// SIMATIC S7-200 project (STEP 7-Micro/WIN), CPU 226 CN REL 02.01

ORGANIZATION_BLOCK 主程序:OB1
TITLE=程序是控制时效炉，用于金属材料热处理
// 
// 风机启动前应确认风压正常。通过风机启动触发鼓风机启动，但鼓风机启动前必须确认东门下限和西门下限已关闭且无故障光报警，以确保通风正常，避免因风压不足影响热处理效果。
// 风机启动后，利用星转角时间切换至风机运行，提供稳定的炉内空气循环。
// 风机运行时，风压开关检测风压状态，若风压异常则触发无风压检测。
// 随后，东门上升和东门下降控制门的位置，但东门上升或东门下降时，必须确认东车运行中为假且未到达东门上限或东门下限，防止门与车碰撞或超出行程。
// 接着，东车前进将材料送入炉内，而东车前进或东车后退时，必须确认东门放松限位为真且无故障光报警，确保通道畅通和运行安全。
// 进入热处理阶段后，加热根据加热信号启动，但加热开始前，必须确认风机运行为真且无超温，避免因通风不足或温度过高损坏材料。加热完成后，系统切换至保温，由保温信号驱动，期间保温必须持续监测超温，若超温则立即停止，防止温度失控影响材料质量。温度控制支持多段工艺，例如通过进入7000系列和第二段温度选择实现不同阶段的升温和保温，必要时通过吸入冷气降温，确保工艺精确性。
// 若检测到电机过热或门故障，系统必须停止风机运行并触发故障声报警，以便工人及时介入排除故障。风压报警时间监测无风压检测，若风压异常则触发故障光报警，提醒操作人员检查通风系统。完成后，西车后退将成品运出，触发周期自动完成标志任务结束。
VAR
i0.0:?;	//  风压开关
i0.1:?;	//  周期自动
i0.2:?;	//  全自动
i0.3:?;	//  风机启动
i0.4:?;	//  风机停止
i0.5:?;	//  东西车、门组合进、退、上、下
i0.6:?;	//  同上
i0.7:?;	//  同上
i1.0:?;	//  东面车、门停止
i1.1:?;	//  东车前进中
i1.2:?;	//  东门锁紧限位
i1.3:?;	//  东门放松限位
i1.4:?;	//  东门上限
i1.5:?;	//  东门下限
i1.6:?;	//  东车前进限
i1.7:?;	//  东车后退限
i2.0:?;	//  西面车、门组合进、退、上、下
i2.1:?;	//  同上
i2.2:?;	//  同上
i2.3:?;	//  西面车、门停止
i2.4:?;	//  西车前进中
i2.5:?;	//  西门锁紧限
i2.6:?;	//  西门放松限
i2.7:?;	//  西门上限
i3.0:?;	//  西门下限
i3.1:?;	//  西车前进限
i3.2:?;	//  西车后退限
i3.3:?;	//  保温信号
i3.4:?;	//  加热信号
i3.5:?;	//  超温
i3.6:?;	//  定时完了信号
i3.7:?;	//  消除报警
i4.0:?;	//  消除铃声
i4.1:?;	//  西车运行中
i4.2:?;	//  东车运行中
i4.3:?;	//  电机过热
i4.4:?;	//  东门上
i4.5:?;	//  东门下
i4.6:?;	//  西门上
i4.7:?;	//  西门下
q0.0:?;	//  风机运行
q0.1:?;	//  保温
q0.2:?;	//  加热
q0.3:?;	//  东车前进
q0.4:?;	//  东车后退
q0.5:?;	//  东门上升
q0.6:?;	//  东门下降
q0.7:?;	//  东门锁紧
q1.0:?;	//  东门放松
q1.1:?;	//  西车前进
q1.2:?;	//  西车后退
q1.3:?;	//  西门上升
q1.4:?;	//  西门下降
q1.5:?;	//  西门锁紧
q1.6:?;	//  西门放松
q1.7:?;	//  定时开始计时
q2.0:?;	//  响铃
q2.1:?;	//  故障声报警
q2.2:?;	//  故障光报警
q2.3:?;	//  周期自动完成
q2.4:?;	//  星形起动
q2.5:?;	//  东门故障
q2.6:?;	//  西门故障
q2.7:?;	//  周期仪表停止
q3.0:?;	//  进入7000系列
q3.1:?;	//  第二段温度选择
q3.2:?;	//  
q3.3:?;	//  停一组加热丝
q3.4:?;	//  吸入冷气
q3.5:?;	//  
q3.6:?;	//  
q3.7:?;	//  
m0.0:?;	//  手动东门锁紧
m0.1:?;	//  手动东门放松
m0.2:?;	//  手动东门上升
m0.3:?;	//  手动东门下降
m0.4:?;	//  手动东门前进
m0.5:?;	//  手动东门后退
m0.6:?;	//  手动西门锁紧
m0.7:?;	//  手动西门放松
m1.0:?;	//  手动西车前进
m1.1:?;	//  手动西车后退
m1.2:?;	//  确定东车在炉内
m1.3:?;	//  确定西车在炉内
m1.4:?;	//  
m1.5:?;	//  手动西门上升
m1.6:?;	//  手动西门下降
m1.7:?;	//  
m2.0:?;	//  计时信号到
m2.1:?;	//  确认台车运行
m2.2:?;	//  确认台车到位
m2.3:?;	//  
m2.4:?;	//  
m2.5:?;	//  
m2.6:?;	//  
m2.7:?;	//  
m3.0:?;	//  循环开始
m3.1:?;	//  确认两台车是否同时行走
m3.2:?;	//  消除声报警
m3.3:?;	//  
m3.4:?;	//  
m3.5:?;	//  
m3.6:?;	//  
m3.7:?;	//  
m4.0:?;	//  二段保温时间到
m4.1:?;	//  
m4.2:?;	//  
m4.3:?;	//  
m5.0:?;	//  鼓风机启动
m5.1:?;	//  东、西门松开故障
m5.2:?;	//  门故障
m5.3:?;	//  不关门启动风机
m5.4:?;	//  东、西门锁故障
m5.5:?;	//  
m5.6:?;	//  
m5.7:?;	//  
m6.0:?;	//  
m6.1:?;	//  
m6.2:?;	//  
m6.3:?;	//  计数复位
m6.4:?;	//  
m6.5:?;	//  二段保温到时
m6.6:?;	//  
m6.7:?;	//  
m8.0:?;	//  
m8.1:?;	//  一段保温到时
m8.2:?;	//  进入时间加温控
m8.3:?;	//  二段到时间
m8.4:?;	//  一段后台车不交换
m8.5:?;	//  二段时间复位
m8.6:?;	//  二段保温
m8.7:?;	//  手动选择
m9.0:?;	//  周期复位
m9.1:?;	//  周期/全自动
m9.2:?;	//  
m9.3:?;	//  无风压检测
m9.4:?;	//  
m9.5:?;	//  
m9.6:?;	//  
m9.7:?;	//  
m10.0:?;	//  0.5秒脉冲
m10.1:?;	//  1分钟计时
m10.2:?;	//  分钟复位
m10.3:?;	//  
m10.4:?;	//  45度开始计时
m10.5:?;	//  7000升温段信号
m10.6:?;	//  二段升温开始
m10.7:?;	//  
m11.0:?;	//  一段停止加热信号
m11.1:?;	//  二段停止加热信号
m11.2:?;	//  一段停止保温信号
m11.3:?;	//  二段停止保温信号
m11.4:?;	//  一段计时开始
m11.5:?;	//  二段计时开始
m11.6:?;	//  
m11.7:?;	//  
t130:?;	//  星转角时间
t131:?;	//  保温误动时间
t132:?;	//  同上
t133:?;	//  加热误动时间
t134:?;	//  同上
t135:?;	//  同上
t136:?;	//  防止风波动
t137:?;	//  确认台车运行
t138:?;	//  两车允许误差
t139:?;	//  出炉报警时间
t140:?;	//  同上
t141:?;	//  同上
t142:?;	//  故障报警时间
t143:?;	//  风压报警时间
t144:?;	//  
t145:?;	//  门故障时间
t146:?;	//  
t147:?;	//  
t163:?;	//  
t164:?;	//  台车故障报警
t165:?;	//  闪动源
t166:?;	//  同上
t167:?;	//  门故障
t168:?;	//  进入7000确认时间
t169:?;	//  一段保温时间到
t170:?;	//  一段后台车不交换确认
t171:?;	//  二段交换台车
t172:?;	//  
t173:?;	//  
c0:?;	//  周期计数
c1:?;	//  .计数
c10:?;	//  一秒钟计数
c11:?;	//  一分钟计数
END_VAR
BEGIN
Network 1 // 网络标题
// 组合开关8421码                                 (东门锁 )
LD     I0.5
AN     I0.6
AN     I0.7
=      M0.0
Network 2
// 组合开关8421码                                ( 东门松)
LDN    I0.5
A      I0.6
AN     I0.7
=      M0.1
Network 3
// 组合开关8421码                                  (东门上)
LD     I0.5
A      I0.6
AN     I0.7
=      M0.2
Network 4
// 组合开关8421码                                    (东门下)
LDN    I0.5
AN     I0.6
A      I0.7
=      M0.3
Network 5
// 组合开关8421码                                   ( 东车进)
LD     I0.5
AN     I0.6
A      I0.7
=      M0.4
Network 6
// 组合开关8421码                                     (东车退)
LDN    I0.5
A      I0.6
A      I0.7
=      M0.5
Network 7
// 组合开关8421码                                   (   西门锁)
LD     I2.0
AN     I2.1
AN     I2.2
=      M0.6
Network 8
// 组合开关8421码                                        (西门松)
LDN    I2.0
A      I2.1
AN     I2.2
=      M0.7
Network 9
// 组合开关8421码                                        ( 西门上)
LD     I2.0
A      I2.1
AN     I2.2
=      M1.5
Network 10
// 组合开关8421码                                          (西门下)
LDN    I2.0
AN     I2.1
A      I2.2
=      M1.6
Network 11
// 组合开关8421码                                              ( 西车进)
LD     I2.0
AN     I2.1
A      I2.2
=      M1.0
Network 12
// 组合开关8421码                                               ( 西车退)
LDN    I2.0
A      I2.1
A      I2.2
=      M1.1
Network 13
// 东车前进限                    西车后退限                ( 东车在炉内)
LDN    I1.6
AN     I3.2
=      M1.2
Network 14
// 东车后退限                      西车后退限                      ( 西车在炉内)
LDN    I1.7
AN     I3.1
=      M1.3
Network 15
// 手动    循环开始     二段时间到   7000系列   西门锁   风机停    西门下  东门下  东门锁  故障  电机热     (风机启动)
// 启动按钮                                                           定时到
// 自保
LDN    M8.7
A      M3.0
O      I0.3
O      M5.0
LDN    M8.6
A      Q3.0
ON     M2.0
ALD
A      I2.5
A      I0.4
A      I3.0
A      I1.5
A      I1.2
AN     Q2.2
AN     I4.3
=      M5.0
Network 16
// 风机启动信号                                         星转三角延时
// 不关门启动风机
LD     M5.0
O      M5.3
TON    T130, +99
Network 17
// 风机启动信号          星转三角延时             三角运行                        (星形运行)
// 不关门启动风机
LD     M5.0
O      M5.3
AN     T130
AN     Q0.0
=      Q2.4
Network 18
// 风机启动信号          星转三角延时              星形运行               (风机运行  )
// 不关门启动风机
LD     M5.0
O      M5.3
A      T130
AN     Q2.4
=      Q0.0
Network 19
// 风机运行                                                                                           保温防震                 (保温防震时间)
LD     Q0.0
AN     T132
TON    T131, +40
Network 20
// 风机运行                      保温信号                                               (保温防震 )
LD     Q0.0
AN     I3.3
AN     Q3.0
LDN    M11.3
A      Q3.0
A      Q3.1
LDN    M11.2
A      Q3.0
AN     Q3.1
OLD
A      Q0.0
OLD
TON    T132, +8
Network 21
// 计时开始                 保温防震时间                  超温                      风压检测           不关门启动风机        (保温)
// 7000系列
// 升温控制
LD     Q1.7
ON     Q3.0
O      M10.5
A      T131
AN     I3.5
A      M9.3
AN     M5.3
=      Q0.1
Network 22
// 加热防震                                              ( 加热防震时间)
LD     T135
TON    T133, +10
Network 23
// 风机启动                       加热防震                                         (加热防震时间)
LD     Q0.0
AN     T135
TON    T134, +40
Network 24
// 加热信号                        7000系列                                          风机启动                                              (加热防震时间)
//  保温信号  
// 
LDN    I3.4
ON     I3.3
AN     Q3.0
LDN    Q3.1
AN     M11.0
LD     Q3.1
AN     M11.1
OLD
A      Q3.0
OLD
A      Q0.0
TON    T135, +20
Network 25
// 升温控制                    加热防震时间            超温                        风压检测              不关门启动风机             (加热)
//  计时开始
// 7000系列
LD     M10.5
O      Q1.7
ON     Q3.0
A      T134
AN     I3.5
A      M9.3
AN     M5.3
=      Q0.2
Network 26
//  加热防震时间              7000 系列                                                一段不交换台车            风机启动            计时开始
// 自保                                                                                                 7000系列
LD     T133
AN     Q3.0
O      Q1.7
LD     Q3.1
A      M11.5
LDN    Q3.1
A      M11.4
OLD
A      Q3.0
OLD
LDN    M8.4
ON     Q3.0
ALD
A      Q0.0
=      Q1.7
Network 27
//    风机启动                     保温信号                超温信号
LD     Q0.0
AN     I3.3
AN     I3.5
AN     C2
=      M6.0
Network 28
LD     I3.3
O      I3.5
AN     C2
=      M6.1
Network 29
LD     M6.1
LD     M6.3
CTU    C2, +1
Network 30
LD     Q1.3
O      Q0.5
=      M6.3
Network 31
// 周期                          定时到               二段到时              确定台车到位                   故障              仃凤机             (计时到)
// 自动                                                              不交换时间
// 自保               
LD     I0.1
O      I0.2
A      I3.6
O      M2.0
LD     M8.6
ON     T170
ALD
AN     M2.2
AN     Q2.2
A      I0.4
=      M2.0
Network 32
// 手动                           西门松                          西门松限                    西门锁紧          (西门放松)
// 自保
// 计时到                       二段到时
LD     M8.7
A      M0.7
O      Q1.6
LD     M2.0
AN     M8.3
OLD
AN     I2.6
AN     Q1.5
=      Q1.6
Network 33
// 风机运行                   风压开关                 失压确认                 停风机                        风压开关                       (失压确认 ) 
// 自保                                                                                                                            (风压)
LD     Q0.0
A      I0.0
O      M9.3
AN     T136
A      I0.4
LPS
AN     I0.0
TON    T136, +600
LPP
=      M9.3
Network 34
// 手动                             东门松                        东门松限                  东门锁                  (  东门松)
// 自保
// 到时                                二段到时
LD     M8.7
A      M0.1
O      Q1.0
LD     M2.0
AN     M8.3
OLD
AN     I1.3
AN     Q0.7
=      Q1.0
Network 35
// 手动      西门上         西门松      西车门仃   西车进      西车退    西门上限     西门下    故障   电热过温      (西门上)
// 自保                            仃风机
// 确定西车在炉            到时                          二段到时
// 周期
LD     M8.7
A      M1.5
LD     Q1.3
A      I0.4
OLD
LD     M1.3
ON     C0
A      M2.0
AN     M8.3
OLD
A      I2.6
A      I2.3
AN     Q1.1
AN     Q1.2
AN     I2.7
AN     Q1.4
AN     Q2.2
AN     I4.3
=      Q1.3
Network 36
// 手动      东门上         西门松      东车门仃   东车进      东车退    东车进       东门下      故障         电热过温      (东门上)
// 自保                            仃风机
// 确定东车在炉            到时                          二段到时
// 周期
LD     M8.7
A      M0.2
LD     Q0.5
A      I0.4
OLD
LD     M1.2
ON     C0
A      M2.0
AN     M8.3
OLD
A      I1.0
A      I1.3
AN     Q0.4
AN     Q0.3
AN     I1.4
AN     Q0.6
AN     Q2.2
AN     I4.3
=      Q0.5
Network 37
// 手动     东车退      东门 车仃止       东门上限    东门上    东门下    东车退限   东车进   故障    电机过热     (东车退)
// 自保                                仃风机
// 确定东车在炉内            到时                          二段到时
LD     M8.7
A      M0.5
LD     Q0.4
A      I0.4
OLD
LD     M1.2
A      M2.0
AN     M8.3
OLD
A      I1.0
A      I1.4
AN     Q0.5
AN     Q0.6
A      I1.7
AN     Q0.3
AN     Q2.2
AN     I4.3
=      Q0.4
Network 38
// 手动     两车退      西门 车仃止       西门上限    西门上    西门下    西车退限   西车进   故障    电机过热     (西车退)
// 确定东车在炉内            到时                          二段到时
// 自保                                仃风机
LD     M8.7
A      M1.0
LD     M1.2
A      M2.0
AN     M8.3
OLD
LD     Q1.1
A      I0.4
OLD
A      I2.3
A      I2.7
AN     Q1.3
AN     Q1.4
A      I3.1
AN     Q1.2
AN     Q2.2
AN     C0
AN     I4.3
=      Q1.1
Network 39
// 手动     东车进    东门 车仃止    东门上限    东门上  东门下  东车进限   东车退      故障    周期   过热          东车退)
// 确定东车在炉内            到时                          二段到时
// 自保                                仃风机
LD     M8.7
A      M0.4
LD     M1.3
A      M2.0
AN     M8.3
OLD
LD     Q0.3
A      I0.4
OLD
A      I1.0
A      I1.4
AN     Q0.5
AN     Q0.6
A      I1.6
AN     Q0.4
AN     Q2.2
AN     C0
AN     I4.3
=      Q0.3
Network 40
// 手动   西车退     西车、门停    西门上限    西门下   西门上    西车退限   西车前进   故障   电机过热   (西车退 )
// 确定东车在炉内            到时                          二段到时
// 自保                                仃风机
LD     M8.7
A      M1.1
LD     M1.3
A      M2.0
AN     M8.3
OLD
LD     Q1.2
A      I0.4
OLD
A      I2.3
A      I2.7
AN     Q1.4
AN     Q1.3
A      I3.2
AN     Q1.1
AN     Q2.2
AN     I4.3
=      Q1.2
Network 41
// 确定东车在炉内  东车后退   西车前进    二段保温到时间    风机停止     到时l旬   (  确认台车运行 )
// 确定西车在炉内         东车前进                 西车后退                  进入7000系列
// 自保                              手动选择                                                                                                  (  确认台车运行 )                  
LD     M1.2
A      Q0.4
A      Q1.1
LD     M1.3
A      Q0.3
A      Q1.2
OLD
LD     M2.1
A      M8.7
OLD
LD     M8.6
ON     Q3.0
ALD
A      I0.4
A      M2.0
TON    T137, +10
=      M2.1
Network 42
// 确定东车在炉内       确认台车运行         风机运行                     风机停止                  (  确认台车到位 )
// 确定西车在炉内
// 自保                              手动选择
LD     M1.2
O      M1.3
A      T137
LD     M2.2
A      M8.7
OLD
AN     Q0.0
A      I0.4
=      M2.2
Network 43
// 东车在炉内   周期   台车到位      东车门停 东门松限  东门下限 东门上升 东车前进 故障 过热 东车后退 东门下降
// 确定西车在炉内
// 手动选择                    手动东门下降
// 东门下降                     风机停止
LD     M1.2
O      M1.3
AN     C0
A      M2.2
LD     M8.7
A      M0.3
LD     Q0.6
A      I0.4
OLD
OLD
A      I1.0
A      I1.3
AN     I1.5
AN     Q0.5
AN     Q0.3
AN     Q2.2
AN     I4.3
AN     Q0.4
=      Q0.6
Network 44
// 东车在炉  周期  台车到位   西门松限  西车门停 西门下限  西门上升 西车前进 西车后退 故障 过热  西门下降
// 确定西车在炉内
// 手动选择                    手动门西下降
// 西门下降                     风机停止
LD     M1.2
O      M1.3
AN     C0
A      M2.2
LD     M8.7
A      M1.6
LD     Q1.4
A      I0.4
OLD
OLD
A      I2.6
A      I2.3
AN     I3.0
AN     Q1.3
AN     Q1.1
AN     Q1.2
AN     Q2.2
AN     I4.3
=      Q1.4
Network 45
// 手动选择              东门锁紧                     东门下限                东门下降              东门锁紧限    东门放松    ( 东门锁紧 )
// 确认台车到位
// 东门锁紧
LD     M8.7
A      M0.0
O      M2.2
O      Q0.7
A      I1.5
AN     Q0.6
AN     I1.2
AN     Q1.0
=      Q0.7
Network 46
// 手动选择                  西门锁紧               西门下限                  西门下降         西门锁紧限        西门放松       ( 西门锁紧 )
// 确认台车到位
// 西门锁紧
LD     M8.7
A      M0.6
O      M2.2
O      Q1.5
A      I3.0
AN     Q1.4
AN     I2.5
AN     Q1.6
=      Q1.5
Network 47
// 消除报警                        消除铃声                  周期自动                风机启动                                                    周期计数 
// 确认台车到位
// 周期复位
LD     I3.7
A      I4.0
O      M2.2
A      I0.1
AN     I0.3
LD     M9.0
CTU    C0, +2
Network 48
// 手动选择                        周期复位
// 风机启动
// 全自动
LD     M8.7
O      I0.3
O      I0.2
=      M9.0
Network 49
// 确认台车到位             东门下限                 西门下限               保温误动时间           风机停止            (  循环开始  )
// 循环开始                     手动选择
LD     M2.2
A      I1.5
A      I3.0
LD     M3.0
AN     M8.7
OLD
AN     T131
A      I0.4
=      M3.0
Network 50
// 西车运行中                     东车运行中           (   确认两台车是否同时行走  )
LD     I4.1
A      I4.2
=      M3.1
Network 51
// 东车运行中           东车前进中              周期自动                 周期计数         确认两台车是否同时行走    两车允许误差
// 东车前进中                  东车运行中                 全自动
// 西车前进中                   西车运行中
//  西车运行中                  西车前进中
LD     I4.2
AN     I1.1
LD     I1.1
AN     I4.2
OLD
LD     I2.4
AN     I4.1
OLD
LD     I4.1
AN     I2.4
OLD
LD     I0.1
O      I0.2
ALD
AN     C0
AN     M3.1
TON    T138, +80
Network 52
// 二段保温                      定时完了信号          二段保温时间到
// 进入7000系列
LD     M8.6
ON     Q3.0
A      I3.6
S      M4.0, 1
Network 53
// 消除报警                      二段保温时间到复位
// 循环开始
// 东车后退
// 西车后退
LD     I3.7
O      M3.0
O      Q0.4
O      Q1.2
R      M4.0, 1
Network 54
// 出炉报警时间                                             出炉报警时间
LD     T140
TON    T139, +20
Network 55
// 二段保温时间到              东车前进            东车后退               西车前进                西车后退         出炉报警时间   (同左)
LD     M4.0
AN     Q0.3
AN     Q0.4
AN     Q1.1
AN     Q1.2
AN     T139
TON    T140, +80
Network 56
// 东车前进                        西车后退                周期计数                 闪动源                                            出炉报警时间
// 东车后退                        西车前进
// 东车后退                         周期计数  
// 西车后退
LD     Q0.3
A      Q1.2
LD     Q0.4
A      Q1.1
OLD
AN     C0
LD     Q0.4
O      Q1.2
A      C0
OLD
A      T165
TON    T141, +10
Network 57
// 出炉报警时间              响铃
LD     T140
=      Q2.0
Network 58
// 进入7000系列                                             热电偶输入口
LD     Q3.0
O      I3.7
MOVW   AIW2, VW418
-I     +0, VW418
Network 59
//      保温                         东车后退              故障光报警
//      加热
//     两车允许误差          周期计数
//    电机过热
LD     Q0.1
O      Q0.2
A      Q0.4
LD     T138
AN     C0
O      I4.3
OLD
S      Q2.2, 1
Network 60
//    消除报警                      消除铃声              故障光报警复位
LD     I3.7
AN     I4.0
R      Q2.2, 1
Network 61
// 故障光报警                                                风压报警时间           消除声报警          故障声报警
// 西门锁紧限                                                  闪动源                 
// 西门故障                                                                                       故障报警时间
// 计数
// 东车前进中                   出炉报警时间
// 西车前进中
// 西车运行中
// 东车运行中
// 出炉报警时间
// 风压报警时间
LD     Q2.2
O      Q2.5
O      Q2.6
O      C1
LD     I1.1
O      I2.4
O      I4.1
O      I4.2
A      T140
OLD
LD     T141
O      T143
OLD
LPS
LD     T143
O      T165
ALD
AN     M3.2
=      Q2.1
LPP
TON    T142, +600
Network 62
// 风机运行                   无风压检测                                          风压报警时间
LD     Q0.0
AN     M9.3
TON    T143, +600
Network 63
// 消除报警                     消除铃声                   鼓风机启动             消除声报警
// 故障报警时间
// 消除声报警
LD     I3.7
AN     I4.0
O      T142
O      M3.2
AN     M5.0
=      M3.2
Network 64
// 周期计数                   周期自动完成
LD     C0
=      Q2.3
Network 65
// 东门下                            东门下降               周期自动                                                门故障时间
// 东门上                           东门上升                全自动
// 西门上                             西门上升
// 西门下                             西门下降
// 西门上升
// 西门下降
// 东门上升
// 东门下降
LDN    I4.5
A      Q0.6
LDN    I4.4
A      Q0.5
OLD
LDN    I4.6
A      Q1.3
OLD
LDN    I4.7
A      Q1.4
OLD
O      Q1.3
O      Q1.4
O      Q0.5
O      Q0.6
LD     I0.1
O      I0.2
ALD
TON    T145, +475
Network 66
// 东车前进中                  周期自动                                                台车故障报警
// 西车前进中                  全自动
// 西车运行中
// 东车运行中
LD     I1.1
O      I2.4
O      I4.1
O      I4.2
LD     I0.1
O      I0.2
ALD
TON    T164, +925
Network 67
// 闪动源                                                         闪动源
LDN    T166
TON    T165, +30
Network 68
// 闪动源                                                              闪动源
LD     T165
TON    T166, +30
Network 69
// 定时完了信号             进入7000系列              周期自动             脉冲上升沿                 东、西门松开故障
// 二段保温                                                               全自动
LD     I3.6
AN     Q3.0
O      M8.6
LD     I0.1
O      I0.2
ALD
EU
S      M5.1, 1
Network 70
// 东门上                             西门上                 东、西门松开故障复位
// 消除报警
LD     I4.4
A      I4.6
O      I3.7
R      M5.1, 1
Network 71
// 星形起动                       东、西门锁故障                                门故障
// 西门上升                       门故障
// 东门上升
LDN    Q2.4
A      M5.4
LDN    Q1.3
ON     Q0.5
A      M5.2
OLD
TON    T167, +100
Network 72
// 西门锁紧                     确认台车到位           脉冲上升沿                 东、西门锁故障
LD     Q1.5
A      M2.2
EU
S      M5.4, 1
Network 73
// 鼓风机启动             东、西门锁故障复位
// 消除报警
LD     M5.0
O      I3.7
R      M5.4, 1
Network 74
// 门故障                            东门放松限位           门故障                       闪动源                   东门故障
// 东、西门锁故障复位      东门锁紧限位
LD     M5.2
AN     I1.3
LD     M5.4
AN     I1.2
OLD
A      T167
A      T165
=      Q2.5
Network 75
// 门故障                            西门放松限位           门故障                       闪动源                   西门故障
// 东、西门锁故障复位      西门锁紧限位
LD     M5.2
AN     I2.6
LD     M5.4
AN     I2.5
OLD
A      T167
A      T165
=      Q2.6
Network 76
// 东车后退                    周期自动完成           周期自动                  周期仪表停止
// 西车后退
// 周期仪表停止
LD     Q0.4
O      Q1.2
A      Q2.3
O      Q2.7
A      I0.1
=      Q2.7
Network 77
// 风机启动                     消除报警                  手动选择                进入7000系列           电机过热             不关门启动风机
// 不关门启动风机            风机停止
LD     I0.3
A      I3.7
LD     M5.3
A      I0.4
OLD
AN     M8.7
A      Q3.0
AN     I4.3
=      M5.3
Network 79
// 周期自动                      进入7000确认时间                            进入7000确认时间
// 进入时间加温控                                  进入时间加温控
LD     I0.1
O      M8.2
AN     T168
TON    T168, +30
=      M8.2
Network 80
// 全自动                   进入时间加温控               手动选择            进入7000系列
// 进入7000系列
LD     I0.2
A      M8.2
O      Q3.0
AN     M8.7
=      Q3.0
Network 81
// 周期自动                          全自动                   手动选择
LDN    I0.1
AN     I0.2
=      M8.7
Network 82
// 计时信号到                  进入7000系列           二段保温                    手动选择              第二段温度选择
// 第二段温度选择
LD     M2.0
A      Q3.0
O      Q3.1
AN     M8.6
AN     M8.7
=      Q3.1
Network 83
//  进入7000系列             定时完了信号          脉冲上升沿           二段时间复位                         一段保温时间到
// 一段保温到时                                                                                                         一段保温到时
LD     Q3.0
A      I3.6
EU
O      M8.1
AN     M8.5
TON    T169, +10
=      M8.1
Network 84
//  一段保温时间到          进入7000系列        定时完了信号             脉冲上升沿          二段时间复位           二段保温
// 二段保温
LD     T169
A      Q3.0
A      I3.6
EU
O      M8.6
AN     M8.5
=      M8.6
Network 85
// 进入7000系列              二段保温                  二段到时间
LD     Q3.0
AN     M8.6
=      M8.3
Network 86
// 计时信号到               进入7000系列     一段后台车不交换确认   二段时间复位                        一段后台车不交换确认 
// 一段后台车不交换                                     二段保温              一段后台车不交换                                     
LD     M2.0
A      Q3.0
O      M8.4
LDN    T170
O      M8.6
ALD
LPS
AN     M8.5
TON    T170, +60
LPP
=      M8.4
Network 87
// 进入7000系列             风压开关                  二段保温                                        二段交换台车
// 二段保温到时                                                                          二段保温到时
LD     Q3.0
AN     Q0.0
O      M6.5
A      M8.6
TON    T171, +10
=      M6.5
Network 88
// 二段交换台车          风压开关                      二段时间复位
// 手动选择
LD     T171
A      Q0.0
O      M8.7
=      M8.5
Network 89
// 0.5秒源                          0.5秒源
LD     SM0.5
=      M10.0
Network 90
// 0.5秒源                           定时开始计时          45度开始计时                                     一秒钟计数
// 1分钟计时
// 手动选择
LD     M10.0
AN     Q1.7
A      M10.4
LD     M10.1
O      M8.7
CTU    C10, +60
Network 91
//   一秒钟计数               1分钟计时
// 分钟复位
LD     C10
O      M10.2
=      M10.1
Network 92
//  一秒钟计数                                            一分钟计数
// 分钟复位
// 手动选择
LD     C10
LD     M10.2
O      M8.7
CTU    C11, +60
Network 93
// 保温误动时间             分钟复位
LD     T132
=      M10.2
Network 94
// 模似量输入口                风机运行             进入7000系列          45度开始计时
// 5度开始计时
LDW>   VW418, +450
A      Q0.0
O      M10.4
A      Q3.0
=      M10.4
Network 95
// 一段升温控制组合                     一分钟计数                    第二段温度选择           进入7000系列          定时开始计时
LDW<   VW418, +800
AW<=   C11, +5
LDW<   VW418, +900
AW>=   C11, +6
AW<=   C11, +13
OLD
LDW<   VW418, +950
AW>=   C11, +13
AW<=   C11, +20
OLD
LDW<   VW418, +970
AW>=   C11, +20
AW<=   C11, +24
OLD
LDW<   VW418, +975
AW>=   C11, +24
AW<=   C11, +25
OLD
LDW<   VW418, +980
AW>=   C11, +26
AW<=   C11, +27
OLD
LDW<   VW418, +985
AW>=   C11, +27
AW<=   C11, +28
OLD
LDW<   VW418, +990
AW>=   C11, +28
AW<=   C11, +29
OLD
LDW<   VW418, +995
AW>=   C11, +29
AW<=   C11, +30
OLD
LDW<   VW418, +1005
AW>=   C11, +30
AW<=   C11, +31
OLD
O      M11.4
AN     Q3.1
LD     M10.6
A      Q3.1
OLD
A      Q3.0
AN     Q1.7
TON    T172, +80
A      T172
=      M10.5
Network 96
// 一段升温控制组合                  一分钟计数                                 一段升温二节
LDW<   VW418, +1010
AW>=   C11, +31
AW<=   C11, +32
LDW<   VW418, +1015
AW>=   C11, +32
AW<=   C11, +33
OLD
LDW<   VW418, +1020
AW>=   C11, +33
AW<=   C11, +34
OLD
LDW<   VW418, +1022
AW>=   C11, +35
AW<=   C11, +37
OLD
LDW<   VW418, +1024
AW>=   C11, +38
AW<=   C11, +40
OLD
LDW<   VW418, +1026
AW>=   C11, +41
AW<=   C11, +43
OLD
LDW<   VW418, +1028
AW>=   C11, +44
AW<=   C11, +46
OLD
LDW<   VW418, +1030
AW>=   C11, +47
AW<=   C11, +50
OLD
LDW<   VW418, +1035
AW>=   C11, +51
AW<=   C11, +53
OLD
LDW<   VW418, +1040
AW>=   C11, +54
AW<=   C11, +57
OLD
LDW<   VW418, +1045
AW>=   C11, +57
AW<=   C11, +59
OLD
LDW<   VW418, +1050
AW>=   C11, +60
OLD
LDW<   VW418, +1050
AW>=   C11, +60
OLD
=      M11.4
Network 97
// 一段升温控制组合               一分钟计数                              第二段温度选择          二段升温开始
LDW<   VW418, +1250
AW<=   C11, +5
LDW<   VW418, +1300
AW>=   C11, +6
AW<=   C11, +12
OLD
LDW<   VW418, +1350
AW>=   C11, +12
AW<=   C11, +16
OLD
LDW<   VW418, +1400
AW>=   C11, +16
AW<=   C11, +17
OLD
LDW<   VW418, +1420
AW>=   C11, +17
AW<=   C11, +18
OLD
LDW<   VW418, +1440
AW>=   C11, +18
AW<=   C11, +19
OLD
LDW<   VW418, +1445
AW>=   C11, +19
AW<=   C11, +20
OLD
LDW<   VW418, +1450
AW>=   C11, +20
AW<=   C11, +21
OLD
LDW<   VW418, +1455
AW>=   C11, +21
AW<=   C11, +22
OLD
LDW<   VW418, +1460
AW>=   C11, +22
AW<=   C11, +23
OLD
LDW<   VW418, +1465
AW>=   C11, +23
AW<=   C11, +24
OLD
LDW<   VW418, +1470
AW>=   C11, +24
AW<=   C11, +25
OLD
LDW<   VW418, +1475
AW>=   C11, +25
AW<=   C11, +26
OLD
LDW<   VW418, +1480
AW>=   C11, +26
AW<=   C11, +27
OLD
LDW<   VW418, +1485
AW>=   C11, +27
AW<=   C11, +28
OLD
LDW<   VW418, +1490
AW>=   C11, +28
AW<=   C11, +29
OLD
LDW<   VW418, +1495
AW>=   C11, +29
AW<=   C11, +30
OLD
LDW<   VW418, +1500
AW>=   C11, +30
OLD
A      Q3.1
=      M10.6
Network 98
// 进入7000系列              热电偶输入口            一段停止加热信号
LD     Q3.0
AW<=   VW418, +1055
=      M11.0
Network 99
// 进入7000系列              热电偶输入口              一段计时开始
LD     Q3.0
AW>=   VW418, +1050
=      M11.4
Network 100
// 进入7000系列              热电偶输入口           一段停止保温信号
LD     Q3.0
AW<=   VW418, +1050
=      M11.2
Network 101
// 进入7000系列              热电偶输入口            二段停止加热信号
LD     Q3.0
AW<=   VW418, +1505
=      M11.1
Network 102
// 进入7000系列              热电偶输入口            二段计时开始
LD     Q3.0
AW>=   VW418, +1500
=      M11.5
Network 103
// 进入7000系列              热电偶输入口            二段停止保温信号
LD     Q3.0
AW>=   VW418, +1505
=      M11.3
Network 104
//                             热电偶输入口             第二段温度选择           进入7000系列         吸入冷气
LDW>=  VW418, +1060
AN     Q3.1
LDW>=  VW418, +1510
A      Q3.1
OLD
A      Q3.0
=      Q3.4
Network 105
//  热电偶输入口         第二段温度选择   进入7000系列         停一组加热丝
LDW>=  VW418, +850
AN     Q3.1
LDW>=  VW418, +1300
A      Q3.1
OLD
A      Q3.0
=      Q3.3
Network 112
// 周期自动                    周期/全自动
// 全自动
LD     I0.1
O      I0.2
=      M9.1
END_ORGANIZATION_BLOCK
